FUNCTION Convert_BOOL_TO_ULINT : Hresult
VAR_INPUT
	in : BOOL;
	out : REFERENCE TO ULINT;
END_VAR
VAR
	converted : ULINT;
END_VAR
VAR CONSTANT
	INCOMPATIBLE : HRESULT := 16#9811070E;
END_VAR

converted := BOOL_TO_ULINT(in);

IF (ULINT_TO_BOOL(converted) <> in) THEN
	Convert_BOOL_TO_ULINT := INCOMPATIBLE;
	RETURN;
END_IF

out := converted;

END_FUNCTION

(* stored: Version 1.1.0.1, ProductVersion 3.1.4024.12
   POU Convert_BOOL_TO_ULINT: Id {e5956cdc-8d20-4e98-bc79-3d655dc46bc4}, SpecialFunc None *)
